// TwinCAT 3 PLC project Untitled1
// ProgramVersion: 3.1.4024.0
// libraries:
//   Tc2_Standard, * (Beckhoff Automation GmbH)
//   Tc2_System, * (Beckhoff Automation GmbH)
//   Tc2_Utilities, * (Beckhoff Automation GmbH)
//   Tc3_Module, * (Beckhoff Automation GmbH)
// project tree:
//   DUTs/ E_EventType.TcDUT, ST_Event.TcDUT
//   / PlcTask.TcTTO
//   POUs/ eventLogger.TcPOU, FB_EventRingBuffer.TcPOU, FB_SaveasCSVFile.TcPOU, I_PersistentEventStorage.TcIO, MAIN.TcPOU, updateDatetimeStamp.TcPOU
// real-time tasks:
//   TASK PlcTask: cycle T#10ms, priority 20, ADS port 350

CONFIGURATION Untitled1
    RESOURCE PLC ON TwinCAT3
        TASK PlcTask(INTERVAL := T#10ms, PRIORITY := 20);
        PROGRAM MAIN WITH PlcTask : MAIN;
    END_RESOURCE
END_CONFIGURATION

// ---- DUTs/E_EventType.TcDUT
{attribute 'qualified_only'}
{attribute 'strict'}
{attribute 'to_string'}

TYPE E_EventType :
(
	Alaram := 0,
	Message := 1
);
END_TYPE

// ---- DUTs/ST_Event.TcDUT
TYPE ST_Event :
STRUCT
	eEventType : E_EventType;
	eEventSeverity : TcEventseverity;
	nEventIdentity : UDINT;
	sEventText : STRING(255);
	dtTimeStamp : DATE_AND_TIME;
END_STRUCT
END_TYPE

// ---- POUs/I_PersistentEventStorage.TcIO
INTERFACE I_PersistentEventStorage

METHOD storeEvent
VAR_INPUT
	stEvent : ST_Event;
END_VAR
END_METHOD

END_INTERFACE

// ---- POUs/MAIN.TcPOU
PROGRAM MAIN
VAR
	//updatetimestamparrayobject : ST_Event;
	//flag : Bool := True;
	eEventType : E_EventType:= E_EventType.Alaram;
	eEventSeverity : TcEventseverity := TcEventSeverity.Error;
	nEventIdentity : UDINT := 143;
	sEventText : STRING(255):= 'Testing out how function blocks work';
	
	flag: BOOL := FALSE;
	SaveCSVFile : FB_SaveasCSVFile;
	EventLogger : eventLogger(SaveCSVFile);
END_VAR

IF flag THEN
	EventLogger.AddEvent(eEventType,eEventSeverity,nEventIdentity, sEventText);
	flag:= FALSE;
END_IF

SaveCSVFile();

END_PROGRAM

// ---- POUs/FB_SaveasCSVFile.TcPOU
FUNCTION_BLOCK FB_SaveasCSVFile IMPLEMENTS I_PersistentEventStorage
VAR_INPUT
END_VAR
VAR_OUTPUT
END_VAR
VAR
	fileopen : FB_FileOpen:= (sPathName:= 'C:\Users\ramak\Downloads\Event Logger\Events.log',nMode:= FOPEN_MODEAPPEND OR FOPEN_MODETEXT);
	fileputs :  FB_FilePuts;
	eWriteState : (fileOpenTrigger, fileOpen, waitForTheEvent,eventWriteTrigger, eventWrite, fileClose, errorHandeling);
	stEventWriteToFile : ST_Event;
	createdCSVString : T_MaxString;
	fbEventRingBuffer : FB_EventRingBuffer;
END_VAR

CASE eWriteState OF
	fileOpenTrigger: 
		fileopen(bExecute:= TRUE);
		eWriteState := fileOpen;
		
	fileOpen :
		fileopen(bExecute:= FALSE);
		IF fileopen.bError THEN
			eWriteState:= errorHandeling;
		ELSIF NOT fileopen.bBusy AND fileopen.hFile <> 0 THEN
			eWriteState := waitForTheEvent;
		END_IF
	waitForTheEvent :
		    IF fbEventRingBuffer.Remove(stEvent => stEventWriteToFile) THEN
        eWriteState := eventWriteTrigger;
    END_IF

	eventWriteTrigger :
		createdCSVString := concatString(stEvent:= stEventWriteToFile);
		fileputs(bExecute:= TRUE, sLine:=createdCSVString, hFile:=fileopen.hFile);
		eWriteState:= eventWrite;
		
	eventWrite:
		fileputs(bExecute:= FALSE);
		IF fileputs.bError THEN
			eWriteState:= errorHandeling;
			ELSIF NOT fileputs.bBusy THEN
				eWriteState:= waitForTheEvent;
		END_IF
		
	errorHandeling :
	//noting
	
END_CASE

METHOD PRIVATE concatString : T_MaxString
VAR_INPUT
	stEvent : REFERENCE TO ST_Event;
END_VAR
VAR
	stringFlag : T_MaxString;
END_VAR
stringFlag:= TO_STRING(stEvent.eEventType);
stringFlag := CONCAT(STR1:= stringFlag, STR2:= TO_STRING(stEvent.eEventSeverity));
stringFlag := CONCAT(STR1:= stringFlag, STR2:= ',');
stringFlag := CONCAT(STR1:= stringFlag, STR2:= TO_STRING(stEvent.dtTimeStamp));
stringFlag := CONCAT(STR1:= stringFlag, STR2:= ',');
stringFlag := CONCAT(STR1:= stringFlag, STR2:= TO_STRING(stEvent.nEventIdentity));
stringFlag := CONCAT(STR1:= stringFlag, STR2:= ',');
stringFlag := CONCAT(STR1:= stringFlag, STR2:= stEvent.sEventText);
stringFlag := CONCAT(STR1:= stringFlag, STR2:= '\n');
concatString := stringFlag;
END_METHOD

METHOD storeEvent
VAR_INPUT
	stEvent	: ST_Event;
END_VAR
VAR
	fbEventRingBuffer : FB_EventRingBuffer;
END_VAR
fbEventRingBuffer.Apend(stEvent:=stEvent);


//IF eWriteState = waitForTheEvent THEN
	//eWriteState := eventWriteTrigger;
	//stEventWriteToFile :=stEvent;
//END_IF
END_METHOD

END_FUNCTION_BLOCK

// ---- POUs/FB_EventRingBuffer.TcPOU
FUNCTION_BLOCK FB_eventRingBuffer
VAR
	bufferRingArray : ARRAY[1..20] OF ST_Event;
	headIndex : INT := 1;
	tailIndex : INT := 1;
	currentPosition : INT := 1;
	
END_VAR
VAR CONSTANT
	ringBufferSize : INT := 20;
END_VAR

METHOD Apend : BOOL
VAR_INPUT
	stEvent : ST_Event;
END_VAR
IF currentPosition >= ringBufferSize THEN
	Apend:= FALSE;
ELSE
	bufferRingArray[headIndex]:= stEvent;		
	headIndex := headIndex+1;
	currentPosition:=currentPosition+1;
	Apend:= True;
END_IF
END_METHOD

METHOD Remove : BOOL
VAR_OUTPUT
	stEvent: ST_Event;
END_VAR
IF currentPosition:=0 THEN
	Remove:= FALSE;
ELSE
	stEvent:= bufferRingArray[currentPosition];
	tailIndex:= tailIndex+1;
	currentPosition:= currentPosition-1;
	Remove:= TRUE;
END_IF
END_METHOD

END_FUNCTION_BLOCK

// ---- POUs/eventLogger.TcPOU
FUNCTION_BLOCK PUBLIC eventLogger
VAR
	eventBuffer : ARRAY[1..Maximum_Size_of_Event_Buffer] OF ST_Event;
	Current_Position : INT := 0;
	
	_PersistantEventStorage : I_PersistentEventStorage;
END_VAR
VAR CONSTANT
	Maximum_Size_of_Event_Buffer : INT := 100;
END_VAR

METHOD PUBLIC AddEvent : BOOL
VAR_INPUT
	eEventType : E_EventType;
	eEventSeverity : TcEventseverity;
	nEventIdentity : UDINT;
	sEventText : STRING(255);
END_VAR
IF NOT IsBufferFull() THEN
	Current_Position:= Current_Position+1;
	eventBuffer[Current_Position].eEventType:= eEventType;
	eventBuffer[Current_Position].eEventSeverity:= eEventSeverity;
	eventBuffer[Current_Position].nEventIdentity:= nEventIdentity;
	eventBuffer[Current_Position].sEventText:= sEventText;
	updateDatetimeStamp(stEvent:= eventBuffer[Current_Position]);
	AddEvent:= TRUE;
ELSE
	AddEvent:= FALSE;
END_IF

_PersistantEventStorage.storeEvent(stEvent := eventBuffer[Current_Position]);
END_METHOD

METHOD FB_init : BOOL
VAR_INPUT
	bInitRetains : BOOL; // if TRUE, the retain variables are initialized (warm start / cold start)
	bInCopyCode : BOOL;  // if TRUE, the instance afterwards gets moved into the copy code (online change)
	iPersistantEventStorage : I_PersistentEventStorage;
END_VAR
_PersistantEventStorage := iPersistantEventStorage;
END_METHOD

METHOD PRIVATE IsBufferFull : BOOL
IF (Current_Position+1) > Maximum_Size_of_Event_Buffer THEN
	IsBufferFull:= TRUE;
ELSE 
	IsBufferFull := FALSE;
END_IF
END_METHOD

END_FUNCTION_BLOCK

// ---- POUs/updateDatetimeStamp.TcPOU
FUNCTION updateDatetimeStamp
VAR_INPUT
	stEvent : REFERENCE TO ST_Event;
	
END_VAR
VAR
	fbgetSystemTime: GETSYSTEMTIME;
	tFilename : T_FILETIME;	
END_VAR

fbgetSystemTime(timeLoDW => tFilename.dwLowDateTime,
	timeHiDW => tFilename.dwHighDateTime);
	
stEvent.dtTimeStamp := FILETIME_TO_DT( filetime:= tFilename);

END_FUNCTION
